{attribute 'qualified_only'}
TYPE E_PlcSystemStatus :
(
	Idle := 0,
	Error := 1,
	Homing := 2,
	Stopping := 3,
	Taring := 4,
	BasicMove := 5,
	ForceMode := 6,
	Pretension := 10,
	PreTestCyclic := 11,
	SingleTest := 20,
	CyclicTest := 21,
	PostTest := 30
);
END_TYPE

(* stored: Version 1.1.0.1, ProductVersion 3.1.4024.15
   DUT E_PlcSystemStatus: Id {79242f3b-aae6-43b4-b3b1-90de0c72bd33} *)
